// Mitsubishi GX Works2 project: b14   PLC: Q02/Q02H

PROGRAM MAIN
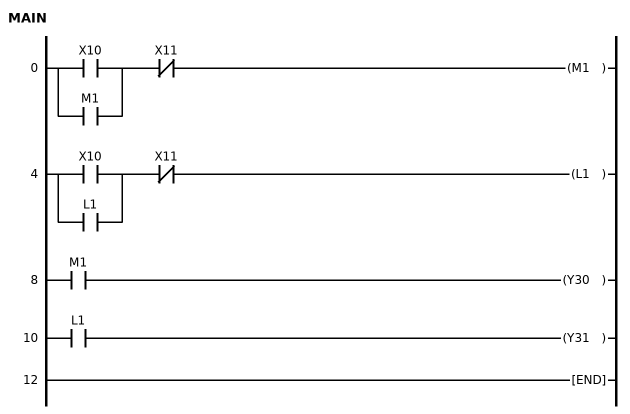
0     LD      X10
      OR      M1
      ANI     X11
      OUT     M1
4     LD      X10
      OR      L1
      ANI     X11
      OUT     L1
8     LD      M1
      OUT     Y30
10    LD      L1
      OUT     Y31
12    END
END_PROGRAM
